TYPE ST_PyAdsConfig :
STRUCT
	sDatabase: STRING;
	sTypeDatabase: STRING;
	sHost: STRING;
	sUser: STRING;
	sPassword: STRING;
END_STRUCT
END_TYPE

(* stored: Version 1.1.0.1, ProductVersion 3.1.4024.2
   DUT ST_PyAdsConfig: Id {ec33ba99-a68a-4559-b930-ae98819283b6} *)
